(* Logix 5000 project; controller AnalogIO_Shared vendor 1 type 14 code 155 rev 36.11; software revision 36.00 *)

TASK MainTask (continuous, watchdog 500 ms) : MainProgram

MODULES
   Local : vendor 1 type 14 code 155 (PointIO 0, rev 36.11)
       : 1734-IE2V (PointIO 2, rev 3.1, Input RPI 80 ms)
       : 1734-OE2V (PointIO 3, rev 3.1, Output RPI 80 ms)
      Discrete_IO : Embedded (PointIO 1, rev 36.11, Output RPI 20 ms)
END_MODULES

PROGRAM MainProgram   (* main routine Elevator *)
VAR
   anyReq : BOOL;
   atFloorTimer : FBD_TIMER;
   currentFloor : DINT;
   dir : DINT;
   dirDOWN : DINT;
   dirNONE : DINT;
   dirUP : DINT;
   doorTimer : FBD_TIMER;
   floor1 : BOOL;
   floor1open : BOOL;
   floor2 : BOOL;
   floor2open : BOOL;
   floor3 : BOOL;
   floor3open : BOOL;
   floor4 : BOOL;
   floor4open : BOOL;
   floorTimer : FBD_TIMER;
   i_DC : ALIAS FOR Local:1:I.Data.14;
   i_DO : ALIAS FOR Local:1:I.Data.15;
   i_E1U : BOOL;
   i_E2D : BOOL;
   i_E2U : BOOL;
   i_E3D : BOOL;
   i_E3U : BOOL;
   i_E4D : BOOL;
   i_F1 : ALIAS FOR Local:1:I.Data.10;
   i_F2 : ALIAS FOR Local:1:I.Data.11;
   i_F3 : ALIAS FOR Local:1:I.Data.12;
   i_F4 : ALIAS FOR Local:1:I.Data.13;
   i_I1 : BOOL;
   i_I2 : BOOL;
   i_I3 : BOOL;
   i_I4 : BOOL;
   lastFloor : DINT;
   lastMove : DINT;
   o_DoorClose : ALIAS FOR Local:1:O.Data.13;
   o_DoorOpen : ALIAS FOR Local:1:O.Data.12;
   o_MD : ALIAS FOR Local:1:O.Data.11;
   o_MU : ALIAS FOR Local:1:O.Data.10;
   ReqAbove : ALIAS FOR Local:1:O.Data.14;
   ReqBelow : ALIAS FOR Local:1:O.Data.15;
   ReqE1U : ALIAS FOR Local:1:O.Data.0;
   ReqE2D : ALIAS FOR Local:1:O.Data.1;
   ReqE2U : ALIAS FOR Local:1:O.Data.2;
   ReqE3D : ALIAS FOR Local:1:O.Data.3;
   ReqE3U : ALIAS FOR Local:1:O.Data.4;
   ReqE4D : ALIAS FOR Local:1:O.Data.5;
   ReqI1 : ALIAS FOR Local:1:O.Data.6;
   ReqI2 : ALIAS FOR Local:1:O.Data.7;
   ReqI3 : ALIAS FOR Local:1:O.Data.8;
   ReqI4 : ALIAS FOR Local:1:O.Data.9;
   s_AtFloor : DINT;
   s_DecideDirection : DINT;
   s_DoorClose : DINT;
   s_DoorOpen : DINT;
   s_Down : DINT;
   s_Up : DINT;
   s_WaitForInput : DINT;
   StateCurrent : DINT;
   StateNext : DINT;
END_VAR

ROUTINE Elevator   (* structured text *)
   doorTimer.Reset := 0;
   floorTimer.Reset := 0;
   atFloorTimer.Reset := 0;
   
   //Floor tracker for floor tags for ignition
   if currentFloor = 1 then floor1 := 1; else floor1 := 0; end_if;
   if currentFloor = 2 then floor2 := 1; else floor2 := 0; end_if;
   if currentFloor = 3 then floor3 := 1; else floor3 := 0; end_if;
   if currentFloor = 4 then floor4 := 1; else floor4 := 0; end_if;
   
   //Latching floor requests from external buttons
   if i_E1U then ReqE1U := 1; end_if;
   if i_E2U then ReqE2U := 1; end_if;
   if i_E2D then ReqE2D := 1; end_if;
   if i_E3U then ReqE3U := 1; end_if;
   if i_E3D then ReqE3D := 1; end_if;
   if i_E4D then ReqE4D := 1; end_if;
   
   //Latching floor requests from internal buttons
   if i_I1 then ReqI1 := 1; end_if;
   if i_I2 then ReqI2 := 1; end_if;
   if i_I3 then ReqI3 := 1; end_if;
   if i_I4 then ReqI4 := 1; end_if;
   
   anyReq := 0;//Force compute of any possible requests each scan
   
   //Combine requests into one latch to indicate whether still WaitForInput or move to DecideDirection
   if ReqE1U then anyReq := 1; end_if;
   if ReqE2U then anyReq := 1; end_if;
   if ReqE2D then anyReq := 1; end_if;
   if ReqE3U then anyReq := 1; end_if;
   if ReqE3D then anyReq := 1; end_if;
   if ReqE4D then anyReq := 1; end_if;
   if ReqI1 then anyReq := 1; end_if;
   if ReqI2 then anyReq := 1; end_if;
   if ReqI3 then anyReq := 1; end_if;
   if ReqI4 then anyReq := 1; end_if;
   
   ReqBelow := 0; //Force compute for these each scan
   ReqAbove := 0;
   
   //Determine if there's a request for above where we are now
   if currentFloor < 2 AND (ReqE2U OR ReqE2D OR ReqI2) then ReqAbove := 1; end_if;
   if currentFloor < 3 AND (ReqE3U OR ReqE3D OR ReqI3) then ReqAbove := 1; end_if;
   if currentFloor < 4 AND (ReqE4D OR ReqI4) then ReqAbove := 1; end_if;
   
   //Determine if there's a request for below where we are now
   if currentFloor > 1 AND (ReqE1U OR ReqI1) then ReqBelow := 1; end_if;
   if currentFloor > 2 AND (ReqE2U OR ReqE2D OR ReqI2) then ReqBelow := 1; end_if;
   if currentFloor > 3 AND (ReqE3U OR ReqE3D OR ReqI3) then ReqBelow := 1; end_if;
   
   //State Machine!
   
   if (s:fs) then
       s_WaitForInput := 0;
       s_DecideDirection := 1;
       s_Up := 2;
       s_Down := 3;
       s_AtFloor := 4;
       s_DoorOpen := 5;
       s_DoorClose := 6;
       dirNONE := 0;
       dirUP := 1;
       dirDOWN := 2;
       floor1 := 1;
       floor2 := 0;
       floor3 := 0;
       floor4 := 0;
       floor1open := 0;
       floor2open := 0;
       floor3open := 0;
       floor4open := 0;
       currentFloor := 1;
       atFloorTimer.PRE := 2000;
       atFloorTimer.TimerEnable := 0;
       floorTimer.PRE := 2000;
       floorTimer.TimerEnable := 0;
       doorTimer.PRE := 1000;
       doorTimer.TimerEnable := 0;
       StateNext := s_WaitForInput;
   end_if;
   
   //Advance state on scan
   StateCurrent := StateNext;
   
   //s_WaitForInput
   if (StateCurrent = s_WaitForInput) then
       dir := dirNONE;
       o_MU := 0;
       o_MD := 0;
       o_DoorOpen := 0;
       o_DoorClose := 0;
   
       //If any buttons pressed then go to s_DecideDirection
       //if (ReqE1U OR ReqE2D OR ReqE2U OR ReqE3D OR ReqE3U OR ReqE4D OR ReqI1 OR ReqI2 OR ReqI3 OR ReqI4) then
       if anyReq then
           StateNext := s_DecideDirection;
       else
           StateNext := s_WaitForInput;
       end_if;
   end_if;
   
   //s_DecideDirection
   if (StateCurrent = s_DecideDirection) then
   	o_MU := 0;
   	o_MD := 0;
   	o_DoorOpen := 0;
   	o_DoorClose := 0;
       // If there is a request at the current floor (and no Requests above or below), serve it immediately and clear requests
       // i.e. All remaining requests are at this floor
       if (currentFloor = 1 AND ReqE1U AND (NOT ReqAbove) AND (NOT ReqBelow)) then
           ReqE1U := 0;
           StateNext := s_DoorOpen;
       else
   		if (currentFloor = 2 AND (ReqE2U OR ReqE2D OR ReqI2) AND (NOT ReqAbove) AND (NOT ReqBelow)) then
           	ReqE2U := 0;
           	ReqE2D := 0;
           	ReqI2 := 0;
           	StateNext := s_DoorOpen;
   		else
       		if (currentFloor = 3 AND (ReqE3U OR ReqE3D OR ReqI3) AND (NOT ReqAbove) AND (NOT ReqBelow)) then
           		ReqE3U := 0;
           		ReqE3D := 0;
           		ReqI3 := 0;
           		StateNext := s_DoorOpen;
   			else
       			if (currentFloor = 4 AND (ReqE4D OR ReqI4) AND (NOT ReqAbove) AND (NOT ReqBelow)) then
           			ReqE4D := 0;
           			ReqI4 := 0;
           			StateNext := s_DoorOpen;
       			else
   			        // Otherwise, follow priority based on current direction or no direction
   			        if (ReqAbove AND dir = dirUP) then
   			            dir := dirUP;
   			            StateNext := s_Up;
   			        else
   			            if (ReqBelow AND dir = dirDOWN) then
   			                dir := dirDOWN;
   			                StateNext := s_Down;
   			            else
   			                if ReqAbove then
   			                    dir := dirUP;
   			                    StateNext := s_Up;
   			                else
   			                    if ReqBelow then
   			                        dir := dirDOWN;
   			                        StateNext := s_Down;
   			                    else
   			                        dir := dirNONE;
   			                        StateNext := s_WaitForInput;
   			                    end_if;
   			                end_if;
   			            end_if;
   			        end_if;
   				end_if;
   			end_if;
   		end_if;
   	end_if;
   end_if;
   
   //s_Up
   if (StateCurrent = s_Up) then
       o_MU := 1;
   	o_MD := 0;
   	o_DoorClose := 0;
   	o_DoorOpen := 0;
       if (floorTimer.ACC = 0 AND (NOT floorTimer.TimerEnable)) then
           floorTimer.TimerEnable := 1;
       end_if;
       if (floorTimer.DN) then
           o_MU := 0;
           floorTimer.TimerEnable := 0;
           floorTimer.Reset := 1;
           lastMove := dirUP;
           StateNext := s_AtFloor;
       else
           StateNext := s_Up;
       end_if;
   end_if;
   
   //s_Down
   if (StateCurrent = s_Down) then
       o_MD := 1;
   	o_MU := 0;
   	o_DoorClose := 0;
   	o_DoorOpen := 0;
       if (floorTimer.ACC = 0 AND (NOT floorTimer.TimerEnable)) then
           floorTimer.TimerEnable := 1;
       end_if;
       if (floorTimer.DN) then
           o_MD := 0;
           floorTimer.TimerEnable := 0;
   		floorTimer.Reset := 1;
           lastMove := dirDOWN;
           StateNext := s_AtFloor;
       else
           StateNext := s_Down;
       end_if;
   end_if;
   
   //s_AtFloor
   if (StateCurrent = s_AtFloor) then
   	o_MD := 0;
   	o_MU := 0;
   	o_DoorClose := 0;
   	o_DoorOpen := 0;
       if (atFloorTimer.ACC = 0 AND (NOT atFloorTimer.TimerEnable)) then
   		if lastMove = dirUP then
               currentFloor := currentFloor + 1;
           else
               if lastMove = dirDOWN then
                   currentFloor := currentFloor - 1;
               end_if;
   		end_if;
           atFloorTimer.TimerEnable := 1;
       end_if;
       if atFloorTimer.DN then
           atFloorTimer.TimerEnable := 0;
   		atFloorTimer.Reset := 1;
           // if currentFloor matches current requests, then open doors
           // Clear UP requests when you've been moving UP and DOWN requests when you've been moving DOWN
           // Always clear internal because people have gotten off of the elevator
   
           // Must do this based on lastMove direction to follow Test Case 1:
           // doors open and close, 1->2 stop doors cont. up, 2->3 stop doors cont. up,
           // 3->4 stop doors go down, 4->3 stop doors cont. down, 3->2 stop doors cont. down, 2->1 stop doors idle
           if (currentFloor = 1 AND (ReqE1U OR ReqI1)) then
               ReqI1 := 0;
   			ReqE1U := 0;
               StateNext := s_DoorOpen;
           else
               if (currentFloor = 2 AND (ReqE2U OR ReqE2D OR ReqI2)) then
                   // only clear Up/Down requests when you were moving in that direction, always clear internal if pressed and you're on that floor
                   if lastMove = dirUP then ReqE2U := 0; end_if;
                   if lastMove = dirDOWN then ReqE2D := 0; end_if;
                   if ReqI2 then ReqI2 := 0; end_if;
                   StateNext := s_DoorOpen;
               else
                   if (currentFloor = 3 AND (ReqE3U OR ReqE3D OR ReqI3)) then
                       if lastMove = dirUP then ReqE3U := 0; end_if;
                       if lastMove = dirDOWN then ReqE3D := 0; end_if;
                       if ReqI3 then ReqI3 := 0; end_if;
                       StateNext := s_DoorOpen;
                   else
                       if (currentFloor = 4 AND (ReqE4D OR ReqI4)) then
                           if lastMove = dirUP then ReqE4D := 0; end_if;
                           if ReqI4 then ReqI4 := 0; end_if;
                           StateNext := s_DoorOpen;
                       else
                           //If no requests for current floor then decide whether to keep going up or down
                           StateNext := s_DecideDirection;
                       end_if;
                   end_if;
               end_if;
           end_if;
       else
           StateNext := s_AtFloor;
       end_if;
   end_if;
   
   //s_DoorOpen
   if (StateCurrent = s_DoorOpen) then
   	o_MU := 0;
   	o_MD := 0;
   	o_DoorClose := 0;
       if (doorTimer.ACC = 0 AND (NOT doorTimer.TimerEnable)) then
           doorTimer.TimerEnable := 1;
       end_if;
       // Floor open tags for door "animation" in ignition
       if currentFloor = 1 then floor1open := 1; else floor1open := 0; end_if;
       if currentFloor = 2 then floor2open := 1; else floor2open := 0; end_if;
       if currentFloor = 3 then floor3open := 1; else floor3open := 0; end_if;
       if currentFloor = 4 then floor4open := 1; else floor4open := 0; end_if;
   	o_DoorOpen := 1;
       if doorTimer.DN then
           o_DoorOpen := 0;
           doorTimer.TimerEnable := 0;
           doorTimer.Reset := 1;
           StateNext := s_DoorClose;
       else
           StateNext := s_DoorOpen;
       end_if;
   end_if;
   
   //s_DoorClose
   if (StateCurrent = s_DoorClose) then
   	o_MU := 0;
   	o_MD := 0;
   	o_DoorOpen := 0;
   	floor1open := 0;
   	floor2open := 0;
   	floor3open := 0;
   	floor4open := 0;
       if (doorTimer.ACC = 0 AND (NOT doorTimer.TimerEnable)) then
           doorTimer.TimerEnable := 1;
       end_if;
   	o_DoorClose := 1;
       if doorTimer.DN then
           o_DoorClose := 0;
           doorTimer.TimerEnable := 0;
           doorTimer.Reset := 1;
           StateNext := s_DecideDirection;
       else
           StateNext := s_DoorClose;
       end_if;
   end_if;
   
   //Store lastFloor in case I end up needing it
   lastFloor := currentFloor;
   
   
   RTOR(doorTimer);
   RTOR(floorTimer);
   RTOR(atFloorTimer);
   
   
END_ROUTINE
END_PROGRAM
